// TwinCAT 3 PLC project main
// ProgramVersion: 3.1.4024.0
// libraries:
//   Tc2_Standard, * (Beckhoff Automation GmbH)
//   Tc2_System, * (Beckhoff Automation GmbH)
//   Tc3_Module, * (Beckhoff Automation GmbH)
// project tree:
//   DUTs/ AmpelState.TcDUT
//   / PlcTask.TcTTO
//   POUs/ MAIN.TcPOU, FB_Ampel.TcPOU
// real-time tasks:
//   TASK PlcTask: cycle T#10ms, priority 20, ADS port 350

CONFIGURATION main
    RESOURCE PLC ON TwinCAT3
        TASK PlcTask(INTERVAL := T#10ms, PRIORITY := 20);
        PROGRAM MAIN WITH PlcTask : MAIN;
    END_RESOURCE
END_CONFIGURATION

// ---- DUTs/AmpelState.TcDUT
{attribute 'qualified_only'}
{attribute 'strict'}
TYPE AmpelState :
(
	Init := 0,
	Red,
	Disabled,
	Red_Yellow,
	Green,
	Yellow
);
END_TYPE

// ---- POUs/MAIN.TcPOU
PROGRAM MAIN
VAR
	clear :		BOOL;
	block :		BOOL;
	disable :	BOOL;
	red :		BOOL;
	yellow :	BOOL;
	green :		BOOL;
	Ampel1 : FB_Ampel;
END_VAR

Ampel1(clear_road:=clear,block_road:=block,disable_system:= disable);
red := Ampel1.red;
yellow := Ampel1.yellow;
green := Ampel1.green;

END_PROGRAM

// ---- POUs/FB_Ampel.TcPOU
FUNCTION_BLOCK FB_Ampel
VAR_INPUT
	clear_road :		BOOL;
	block_road :		BOOL;
	disable_system :	BOOL;
END_VAR
VAR_OUTPUT
	red :				BOOL;
	yellow :			BOOL;
	green :				BOOL;
END_VAR
VAR
	actualState	:		AmpelState := AmpelState.Init;
	timer : 			TON;
	yellowred_lightDuration : 	TIME := T#2S;
	yellow_lightDuration : 		TIME := T#5S;
	blink_lightDuration : 		TIME := T#0.5S;
END_VAR










CASE actualState OF
	AmpelState.Init:
	actualState := AmpelState.Red;
	;
	AmpelState.Red:
	red := TRUE;
	yellow := FALSE;
	green := FALSE;
	IF disable_system THEN
		actualState := AmpelState.Disabled;
	ELSE 
		IF clear_road THEN
			actualState := AmpelState.Red_Yellow;
		END_IF
	END_IF
	;
	AmpelState.Disabled:
	red := FALSE;
	green := FALSE;
	timer(IN:= TRUE,PT:=blink_lightDuration);
	IF timer.Q THEN
		timer(IN:=FALSE, PT:= blink_lightDuration);
		yellow := NOT yellow;
	END_IF
	IF NOT disable_system THEN
		actualState := AmpelState.Red;
	END_IF
	;
	AmpelState.Red_Yellow:
	red := TRUE;
	yellow := TRUE;
	green := FALSE;
	timer(IN:= TRUE,PT:=yellowred_lightDuration);
	IF timer.Q THEN
		timer(IN:=FALSE, PT:= yellowred_lightDuration);
		actualState := AmpelState.Green;
	END_IF
	;
	AmpelState.Green:
	red := FALSE;
	yellow := FALSE;
	green := TRUE;
	IF block_road THEN
		actualState := AmpelState.Yellow;
	END_IF
	;
	AmpelState.Yellow:
	red := FALSE;
	yellow := TRUE;
	green := FALSE;
	timer(IN:= TRUE,PT:=yellow_lightDuration);
	IF timer.Q THEN
		timer(IN:=FALSE, PT:= yellow_lightDuration);
		actualState := AmpelState.Red;
	END_IF
	;
END_CASE

END_FUNCTION_BLOCK
